// TIA Portal V20 export
DATA_BLOCK "Instance_FB_Electrical_Current_Test_DB"   // DB106
// stored: AutoNumber false, InstanceOfName FB_Electrical_Current_Test, InstanceOfType FB
"FB_Electrical_Current_Test"
   // VAR_INPUT
   //    Star_Functional_Test : Bool;
   //    Reset_Functional_Test : Bool;
   //    Electrical_Current_Read_UInt : UInt;
   //    In_Test_Parameters : "IO_Device_Test_Parameters";
   // END_VAR
   // VAR_OUTPUT
   //    Electrical_Current_Test_Approved : Bool;
   // END_VAR
   // VAR
   //    Timer_Delay_Read_Current { S7_SetPoint := 'True'} : TON_TIME;
   //    Timer_Delay_Reset { S7_SetPoint := 'True'} : TON_TIME;
   // END_VAR
BEGIN
END_DATA_BLOCK
